FUNCTION_BLOCK EmergencySystem

// Do nothing here. Function block was split into sub-methods!

METHOD PUBLIC AlarmSystem

VAR_INPUT			// Input variables
	ClearButton : BOOL;
	EmergencyButton : BOOL;
END_VAR

VAR					// Internal (instance) variables
	bIsInitialized : BOOL;
END_VAR
IF NOT bIsInitialized THEN	// Initialization, since functions can't run in top pane
	bIsInitialized := TRUE;
	gAL.fbAlarm.CreateEx(TC_Events.TankAlarmEvent.Emergency, TRUE, 0);
END_IF

IF NOT EmergencyButton THEN
	gAL.fbAlarm.Raise(0); // 0 -> Current time
END_IF

IF (ClearButton AND gAL.fbAlarm.bRaised) THEN
	gAL.fbAlarm.Clear(0, TRUE);	// .Clear(CurrentTime, ConfirmAlarm)
END_IF
END_METHOD

METHOD PUBLIC EmergencyLogic

VAR_INPUT			// Input variables
	EmergencyButton : BOOL;
END_VAR

VAR_IN_OUT			// Pass by reference variables
	MotorState : BOOL;
	FV1percent : INT;
	LV1percent : INT;
	LV2percent : INT;
	LV3percent : INT;
END_VAR
	// Button check, inverted
IF NOT EmergencyButton THEN
	MotorState := FALSE;
	FV1percent := 100;
	LV1percent := 100;
	LV2percent := 100;
	LV3percent := 100;
END_IF

	// Temperature check TBA
	
	// Pressure check TBA
END_METHOD

END_FUNCTION_BLOCK

(* stored: Version 1.1.0.1, ProductVersion 3.1.4024.12
   POU EmergencySystem: Id {ff8af221-7c2c-420a-82d2-c72830098d6c}, SpecialFunc None
   Method AlarmSystem: Id {56e1c5cb-b349-4390-aac6-4099d16cd53c}
   Method EmergencyLogic: Id {209a9a5c-22e1-4953-85b4-acb5c95ad300} *)
